PROGRAM SafetyEnding
VAR
END_VAR

IF Automatic.RotationPositionCurrent >= 570 AND NOT IO.ButtonLowerLeft THEN
	IO.MotorRotation := 0;
END_IF

IF IO.EndRotationSensor THEN	// intermediate reset for accuracy
	Automatic.RotationPositionCurrent := 0;
END_IF

END_PROGRAM

(* stored: Version 1.1.0.1, ProductVersion 3.1.4024.13
   POU SafetyEnding: Id {8bf2167f-22d8-4543-8367-d7ef70615958}, SpecialFunc None *)
